ABB RobotStudio station: SolutionPFC.rspag

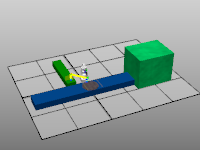
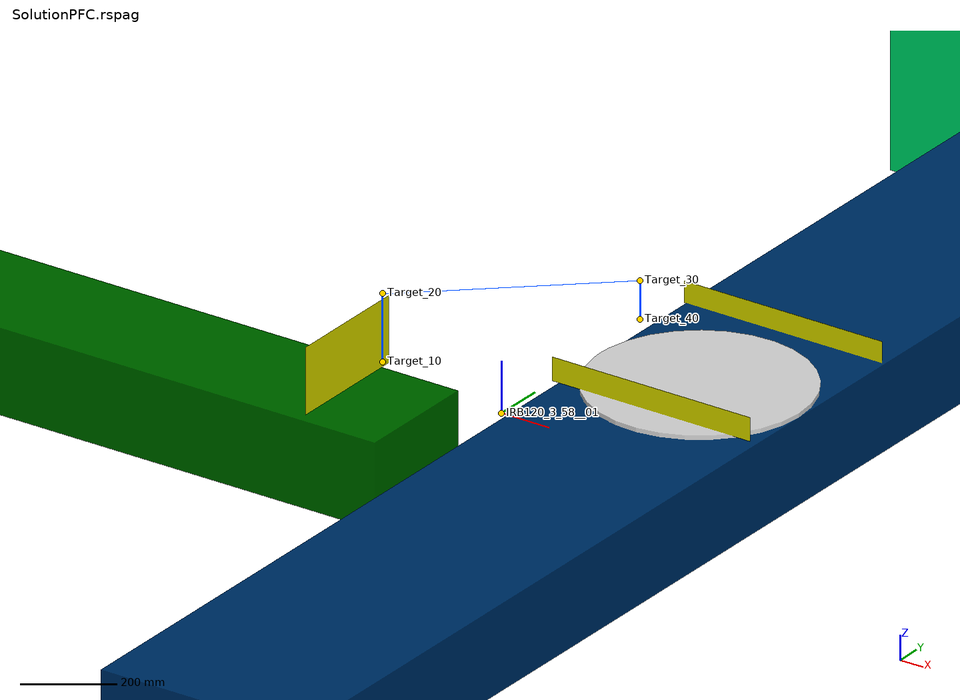
[picture v1: parts stored in the station drawn from their meshes, with robot base, taught points and paths (robot models come from the ABB library and are not in the file)]
--- station ---
Station SolutionPFC (saved by RobotStudio 21.2.9526.0)
Controller Controlador1
  mechanical unit ROB_1: IRB120_3_58__01, 6 joints, base frame (0, 0, 0) mm
Layout (positions relative to the parent item):
  - IRB120_3_58__01 [mechanism, from Robots\IRB120_3_58_G_01.rslib] at (0, 0, 0) mm; joint values [-0.3305, -0.027, -0.2549, 0.2141, 1.2237, -0.3379] (rad or m)
  - Componente inteligente_PALETS [smart component]
      signals: DI COMIENZOPALET, DI ROTAR, DO ROTADO, DI ELEVARROTAR, DI BAJARROTAR, DI CINTAON
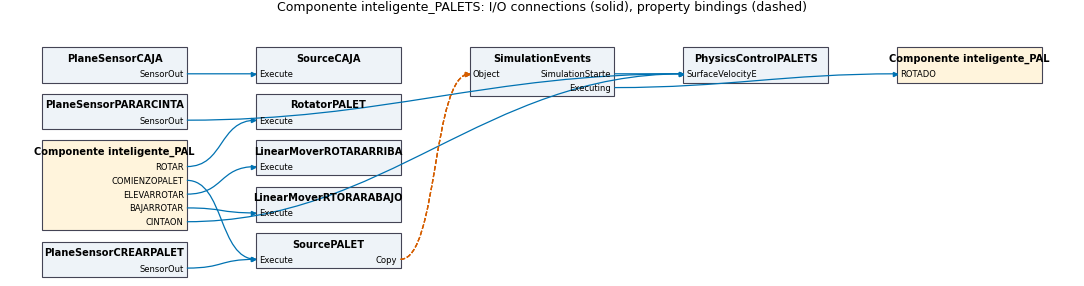
      connections:
        PlaneSensorCAJA.SensorOut -> SourceCAJA.Execute
        PlaneSensorPARARCINTA.SensorOut -> PhysicsControlPALETS.SurfaceVelocityEnabled
        SimulationEvents.SimulationStarted -> PhysicsControlPALETS.SurfaceVelocityEnabled
        Componente inteligente_PALETS.ROTAR -> RotatorPALET.Execute
        Componente inteligente_PALETS.COMIENZOPALET -> SourcePALET.Execute
        PlaneSensorCREARPALET.SensorOut -> SourcePALET.Execute
        RotatorCILINDRO.Executing -> Componente inteligente_PALETS.ROTADO
        Componente inteligente_PALETS.ELEVARROTAR -> LinearMoverROTARARRIBA.Execute
        Componente inteligente_PALETS.BAJARROTAR -> LinearMoverRTORARABAJO.Execute
        Componente inteligente_PALETS.CINTAON -> PhysicsControlPALETS.SurfaceVelocityEnabled
        SourcePALET.Copy => Rotator2.Object
        SourcePALET.Copy => RotatorCILINDRO.Object
        SourcePALET.Copy => MoveAlongCurve.Object
    - CINTA PALET [part], size 512 x 3309.5 x 208.6 mm
    - PALET [part] at (503.22, -1493.81, 203.88) mm, size 350 x 350 x 50 mm
    - ROTAR1 [part] at (0, 0, 10.1) mm, size 500 x 499.3 x 200 mm
    - SourcePALET [smart component, from Components\Source.rslib]
        properties: Source=PALET; Copy=(none); Parent=(none); Position=[0.503219 -1.493811 0.203879]; Orientation=[0 0 0]; Transient=true; PhysicsBehavior=3
    - PlaneSensorPARARCINTA [smart component, from Components\PlaneSensor.rslib] at (0, -270, 15) mm
        properties: Origin=[0.25 0.095 0.2]; Axis1=[0.5 0 0]; Axis2=[0 0 0.055]; SensedPart=(none)
      - _sensorPart_ [part], size 500 x 0 x 55 mm
    - PhysicsControlPALETS [smart component, from Components\PhysicsControl.rslib]
        properties: Object=CINTA PALET; Behavior=1; SurfaceVelocity=0.1
    - RotatorPALET [smart component, from Components\Rotator2.rslib]
        properties: Object=ROTAR1; CenterPoint=[0.5 0 0.2]; Axis=[0 0 1]; Angle=1.5707963267949; Duration=2; Reference=Global; ReferenceObject=(none)
    - PlaneSensorCREARPALET [smart component, from Components\PlaneSensor.rslib]
        properties: Origin=[0.25 0.3 0.205]; Axis1=[0.5 0 0]; Axis2=[0 0 0.05]; SensedPart=(none)
      - _sensorPart_ [part], size 500 x 0 x 50 mm
    - LinearMoverROTARARRIBA [smart component, from Components\LinearMover2.rslib]
        properties: Object=ROTAR1; Direction=[0 0 0.001]; Distance=0.01; Duration=1; Reference=Global; ReferenceObject=(none)
    - LinearMoverRTORARABAJO [smart component, from Components\LinearMover2.rslib]
        properties: Object=ROTAR1; Direction=[0 0 -0.001]; Distance=0.01; Duration=1; Reference=Global; ReferenceObject=(none)
  - Componente inteligente_CAJAS [smart component]
      signals: DO CAJAENPOSICION, DI COMIENZOCAJA, DI ATACHERCAJAS, DI DETACHERCAJA, DI SOURCEPROCESO, DI CINTAON
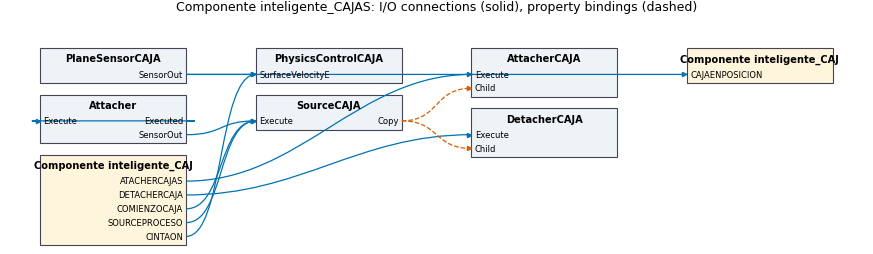
      connections:
        PlaneSensorCAJA.SensorOut -> PhysicsControlCAJA.SurfaceVelocityEnabled
        Attacher.Executed -> Detacher.Execute
        PlaneSensorCAJA.SensorOut -> Componente inteligente_CAJAS.CAJAENPOSICION
        Componente inteligente_CAJAS.ATACHERCAJAS -> AttacherCAJA.Execute
        Componente inteligente_CAJAS.DETACHERCAJA -> DetacherCAJA.Execute
        Componente inteligente_CAJAS.COMIENZOCAJA -> SourceCAJA.Execute
        PlaneSensor.SensorOut -> SourceCAJA.Execute
        Componente inteligente_CAJAS.SOURCEPROCESO -> SourceCAJA.Execute
        Componente inteligente_CAJAS.CINTAON -> PhysicsControlCAJA.SurfaceVelocityEnabled
        SourceCAJA.Copy => AttacherCAJA.Child
        SourceCAJA.Copy => DetacherCAJA.Child
    - PlaneSensorCAJA [smart component, from Components\PlaneSensor.rslib] at (0, 0, 15) mm
        properties: Origin=[-0.075 -0.6 0.2]; Axis1=[0 0.3 0]; Axis2=[0 0 0.155]; SensedPart=(none)
      - _sensorPart_ [part], size 0 x 300 x 155 mm
    - SourceCAJA [smart component, from Components\Source.rslib]
        properties: Source=CAJA; Copy=(none); Parent=(none); Position=[-1.3125 -0.4475 0.2]; Orientation=[0 0 0]; Transient=true; PhysicsBehavior=3
    - CAJA [part] at (-1251.41, -447.5, 200) mm, size 175 x 175 x 100 mm
    - CINTA CAJA [part], size 1500 x 300 x 200 mm
    - PhysicsControlCAJA [smart component, from Components\PhysicsControl.rslib]
        properties: Object=CINTA CAJA; Behavior=1; SurfaceVelocity=0.1
    - AttacherCAJA [smart component, from Components\Attacher.rslib]
        properties: Parent=MyTool; Flange=0; Child=(none); Mount=false; Offset=[0 0 0]; Orientation=[0 0 0]
    - DetacherCAJA [smart component, from Components\Detacher.rslib]
        properties: Child=(none); KeepPosition=true
  - MyTool [mechanism, from Training Objects\myTool.rslib] at (293.39, -85.46, 654.41) mm, rotated rx 180 ry 38 rz 180 deg
  - CAJABORRAR [part], size 1000 x 1200 x 1000 mm
  - RAMPA [part] at (-500, 0, -200) mm, size 500 x 200 x 200 mm
Attachment: CINTA PALET is attached to CINTA CAJA
Attachment: MyTool is attached to IRB120_3_58__01 / Link6
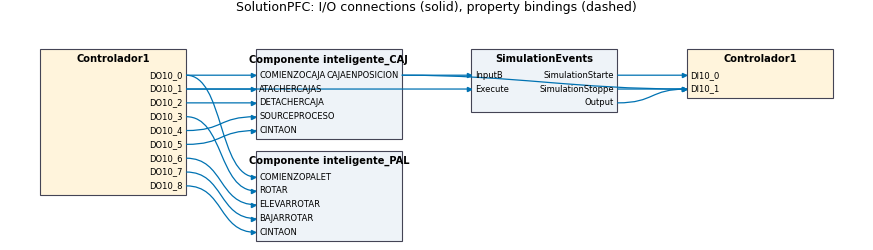
Station logic (signal -> signal, property => property):
  SimulationEvents.SimulationStarted -> Controlador1.DI10_0
  SimulationEvents.SimulationStopped -> Controlador1.DI10_1
  Controlador1.DO10_0 -> Componente inteligente_PALETS.COMIENZOPALET
  Controlador1.DO10_0 -> Componente inteligente_CAJAS.COMIENZOCAJA
  Componente inteligente_CAJAS.CAJAENPOSICION -> LogicGate.InputB
  LogicGate.Output -> Controlador1.DI10_1
  Controlador1.DO10_1 -> Attacher_3.Execute
  Controlador1.DO10_1 -> Componente inteligente_CAJAS.ATACHERCAJAS
  Controlador1.DO10_2 -> Componente inteligente_CAJAS.DETACHERCAJA
  Controlador1.DO10_3 -> Componente inteligente_PALETS.ROTAR
  Controlador1.DO10_4 -> Componente inteligente_CAJAS.SOURCEPROCESO
  Controlador1.DO10_5 -> Componente inteligente_CAJAS.CINTAON
  Componente inteligente_CAJAS.CAJAENPOSICION -> Controlador1.DI10_1
  Controlador1.DO10_6 -> Componente inteligente_PALETS.ELEVARROTAR
  Controlador1.DO10_7 -> Componente inteligente_PALETS.BAJARROTAR
  Controlador1.DO10_8 -> Componente inteligente_PALETS.CINTAON

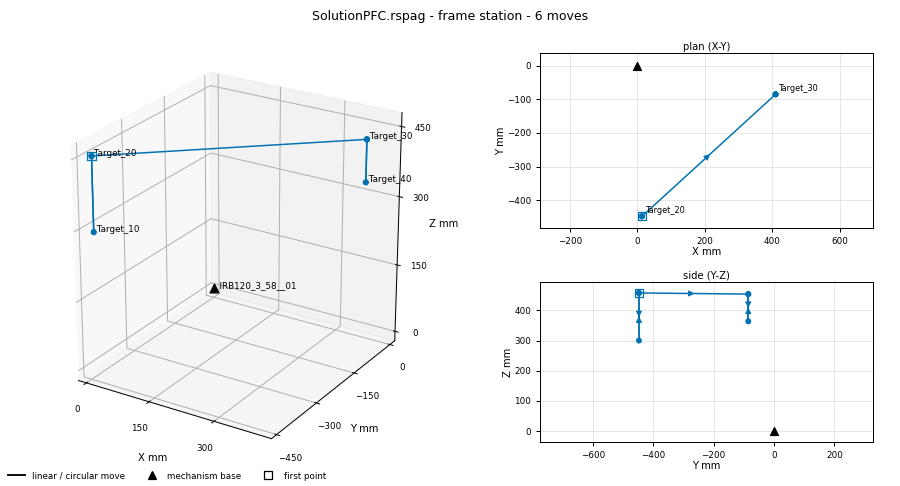
[picture p0: tool path of SolutionPFC.rspag in frame station, 6 of 6 moves have a stored position in this frame; points joined in program order, loops and branches not executed]
--- Backups/Controlador1/RAPID/TASK1/PROGMOD/CalibData.mod ---
MODULE CalibData
    PERS tooldata MyTool:=[TRUE,[[31.7926,0,229.639],[0.945519,0,0.325568,0]],[1,[0,0,1],[1,0,0,0],0,0,0]];
ENDMODULE

--- Backups/Controlador1/RAPID/TASK1/PROGMOD/Module1.mod ---
MODULE Module1
    CONST robtarget Target_10:=[[13.388999591,-447.500002109,299.999996303],[0.000000033,0.707106785,0.707106778,-0.000000023],[-1,0,-1,0],[9E+09,9E+09,9E+09,9E+09,9E+09,9E+09]];
    CONST robtarget Target_20:=[[13.389012212,-447.500004318,457.757996303],[-0.000000033,0.707106785,0.707106778,-0.000000023],[-1,0,-1,0],[9E+09,9E+09,9E+09,9E+09,9E+09,9E+09]];
    CONST robtarget Target_30:=[[409.720015522,-85.464008257,453.878969425],[-0.00000004,0.000000005,1,0.000000007],[-1,0,-1,0],[9E+09,9E+09,9E+09,9E+09,9E+09,9E+09]];
    CONST robtarget Target_40:=[[409.720008322,-85.464006997,363.878969425],[-0.00000004,0.000000005,1,0.000000007],[-1,0,-1,0],[9E+09,9E+09,9E+09,9E+09,9E+09,9E+09]];
    VAR num cont:=0;

    PROC main()
    RESET DO10_6;
    RESET DO10_7;
    IF MARCHAPARO=1 THEN
        SET DO10_0;
        SET DO10_5;
        SET DO10_8;
        ENDIF
    IF MARCHAPARO=0 THEN
        RESET DO10_5;
        RESET DO10_8;
        RESET DO10_0;
        ENDIF
    IF DI10_1=1 THEN
        Path_10;
        ENDIF
    ENDPROC
    PROC Path_10()
        WAITTIME 5;
        RESET DO10_5;
        WAITTIME 3;
        RESET DO10_8;
        SET DO10_6;
        etiqueta1:
        WAITTIME 10;
        MoveL Target_20,v200,fine,MyTool\WObj:=wobj0;
        MoveL Target_10,v200,fine,MyTool\WObj:=wobj0;
        SET DO10_1;
        MoveL Target_20,v200,fine,MyTool\WObj:=wobj0;
        RESET DO10_5;
        MoveL Target_30,v200,fine,MyTool\WObj:=wobj0;
        MoveL Target_40,v200,fine,MyTool\WObj:=wobj0;
        SET DO10_2;
        SET DO10_4;
        SET DO10_3;
        WAITTIME 3;
        SET DO10_5;
        MoveL Target_30,v200,z100,MyTool\WObj:=wobj0;
        RESET DO10_1;
        RESET DO10_2;
        RESET DO10_3;
        RESET DO10_4;
        RESET DO10_6;
        cont:=cont+1;
        IF cont<4 GOTO
        etiqueta1;
        cont:=0;
        WAITTIME 1;
        SET DO10_7;
        WAITTIME 2;
        SET DO10_8;

    ENDPROC
    ENDMODULE

--- Backups/Controlador1/SYSPAR/EIO.cfg ---
EIO:CFG_1.0:6:1::
#
INDUSTRIAL_NETWORK:

      -Name "DeviceNet" -Label "DeviceNet Master/Slave Network" -Address "2"
#
DEVICENET_DEVICE:

      -Name "d652" -VendorName "ABB Robotics" -ProductName "24 VDC I/O Device"\
      -Label "DSQC 652 24 VDC I/O Device" -Address 10 -ProductCode 26\
      -DeviceType 7 -ConnectionType "COS" -OutputSize 2 -InputSize 2
#
DEVICENET_INTERNAL_DEVICE:

      -Name "DN_Internal_Device" -VendorName "ABB Robotics"\
      -ProductName "DeviceNet Internal Slave Device"
#
EIO_SIGNAL:

      -Name "MARCHAPARO" -SignalType "DI" -Device "d652" -DeviceMap "0"

      -Name "DI10_1" -SignalType "DI" -Device "d652" -DeviceMap "1"

      -Name "DI10_2" -SignalType "DI" -Device "d652" -DeviceMap "2"

      -Name "DI10_3" -SignalType "DI" -Device "d652" -DeviceMap "3"

      -Name "DO10_0" -SignalType "DO" -Device "d652" -DeviceMap "0"

      -Name "DO10_1" -SignalType "DO" -Device "d652" -DeviceMap "1"

      -Name "DO10_2" -SignalType "DO" -Device "d652" -DeviceMap "2"

      -Name "DO10_3" -SignalType "DO" -Device "d652" -DeviceMap "3"

      -Name "DO10_4" -SignalType "DO" -Device "d652" -DeviceMap "4"

      -Name "DO10_5" -SignalType "DO" -Device "d652" -DeviceMap "5"

      -Name "DO10_6" -SignalType "DO" -Device "d652" -DeviceMap "6"

      -Name "DO10_7" -SignalType "DO" -Device "d652" -DeviceMap "7"

      -Name "DO10_8" -SignalType "DO" -Device "d652" -DeviceMap "8"

      -Name "DO10_9" -SignalType "DO" -Device "d652" -DeviceMap "9"
